Staubli VAL3: TcpStrRec.dtx

public num nCtrl = 51
public num nFeedback = 52
public num nS8 = 120
public num nV8 = 3
sio sock = {link=Socket\socket1}
public sio socket = {link=Socket\socket1}
string datarec
